{attribute 'GeneratedUsingTerminal: EK1100-0000-0018'}
{attribute addProperty BoxType "EK1100-0000-0018"}
{attribute addProperty Id "Beckhoff_EQ3xxxEK1122Beckhoff_EQ3xxxEK1122_D38136B7718"}
{attribute addProperty CRC "2122666291"}
{attribute addProperty Size "718"}
TYPE Beckhoff_EQ3xxx_7E855133 EXTENDS EK1100_AB5A9467 :
STRUCT
	{attribute addProperty Name "Beckhoff_EQ3xxxEK1122"}
	{attribute addProperty PreviousPort "Beckhoff EQ3xxx : B"}
	Beckhoff_EQ3xxxEK1122 : Beckhoff_EQ3xxxEK1122_D38136B7;
END_STRUCT
END_TYPE

(* stored: Version 1.2.0.0, ProductVersion 3.1.4024.9
   DUT Beckhoff_EQ3xxx_7E855133: Id {552b4b20-94bb-4cca-9a74-f3c528dbfe06} *)
